DATA_BLOCK "GeneralDebug"
{ S7_Optimized_Access := 'TRUE' }
VERSION : 0.1
NON_RETAIN
// ATTRIBUTES
// AUTO_NUMBER = True
// BLOCK_NUMBER = 1
// END_ATTRIBUTES
   VAR
      Debug : Array[1..99] of Bool;
   END_VAR


BEGIN

END_DATA_BLOCK

